(* CODESYS project Pi_Serial_FB_10.project

Project tree, tasks and I/O mapping:
  Device : CODESYS Control for Raspberry Pi SL, 3S - Smart Software Solutions GmbH, version 3.5.12.10
    application Application
      libraries: Standard, * (System); CAA SerialCom, 3.5.12.0 (CAA Technical Workgroup); CAA Types Extern, 3.5.10.0 (CAA Technical Workgroup); CAA Memory, 3.5.12.0 (CAA Technical Workgroup)
      task MainTask (cyclic, interval t#20ms, priority 1) calls PLC_PRG
      task VISU_TASK (cyclic, interval 100 ms, priority 31) calls VisuElems.Visu_Prg
      program PLC_PRG [SFC]: _aInit_active, write_active, read_active, disconnect_active, error_active, Set_COM_active
      visualisation Visualization
      global variables GVL
    SoftMotion General Axis Pool
    I²C
    SPI
      SPI_master : SPI master, 3S - Smart Software Solutions GmbH, version 1.0.0.0
        PiXtend : PiXtend, Qube Solutions UG, version 1.0.0.10
            output Application.GVL.xDO0 : BOOL  // RelayOut.Bit0
            output Application.GVL.byUCControl : BYTE  // CtrlUC
            input  Application.GVL.byUCVersionL : BYTE  // ucVersion_Low
            input  Application.GVL.byUCVersionH : BYTE  // ucVersion_High
            input  Application.GVL.byUCStatus : BYTE  // ucStatus
            unmapped channels: DigIn, GpioIn, AI0, AI1, AI2, AI3, AI0 Raw, AI1 Raw, AI2 Raw, AI3 Raw, Temp0, Temp1, Temp2, Temp3, Humidity0, Humidity1, Humidity2, Humidity3, DigOut, GpioOut, RelayOut, Pwm0, Pwm1, CtrlPwm0, CtrlPwm1, CtrlPwm2, CtrlGpio, CtrlAi0, CtrlAi1, AI Jumpers, DHT11/22
    GPIOs_A_B : GPIOs A/B, 3S - Smart Software Solutions GmbH, version 3.5.11.0
        output rpi_gpio24 : BOOL  // digital outputs (GPIO0..GPIO31).Bit24
        unmapped channels: digital inputs (GPIO0..GPIO31), digital outputs (GPIO0..GPIO31)
    Onewire
    Camera device
      <Empty>
  libraries: VisuSymbols, 3.5.10.0 (System)
  text list GlobalTextList
*)

// Device/Application/GVL
{attribute 'qualified_only'}
VAR_GLOBAL	

	//Digital Outputs
	xDO0: BOOL;
	//Status
	byUCStatus: BYTE;
	byUCVersionL: BYTE;
	byUCVersionH: BYTE;
	//Control
	byUCControl: BYTE;	
END_VAR

// Device/Application/PLC_PRG
PROGRAM PLC_PRG
VAR
	//Visu Variables
	xBtnClear		: BOOL := FALSE;
	xClearAll		: BOOL;	// flag to clear all
	
	//Current State
	iState : INT := 0;

	(* Settings to communicate with the COM Port *)
	aCom1Params : ARRAY [1..7] OF COM.PARAMETER; 
	
	hCom	: CAA.HANDLE; (* handle of the port*)
	como1 	: COM.Open;
	comc1 	: COM.Close;
	comw1 	: COM.Write;
	comr1 	: COM.Read;	
	
	
	sWrite 	: STRING;
	szRead 	: CAA.SIZE;
	uiRead	: UINT;
	
	bReadBuffer	: ARRAY [1..255] OF BYTE; (*Used to read data from the serial port*)
	sReadText	: STRING;
	
	bWriteBuffer: ARRAY [1..255] OF BYTE; (*Used to write data to the serial port*)
	szWrite		: CAA.SIZE;
	
	xReadSuccess	: BOOL;
	xWriteSuccess	: BOOL;
	
	// errors
	xCom1OpenError 	: BOOL;
	xCom1WriteError : BOOL;
	xCom1ReadError 	: BOOL;
	iError			: INT;
	errWrite 		: INT;
	errRead 		: INT;
	Bar				: INT;
	Bar_Temp		: INT;
	
	tTimer			: TON;
	
	sSend 		: STRING(255);	// send message
	sStatus 	: STRING(25);	// status message
	
	//arsReceived : ARRAY[0..1,0..10000] OF STRING(255);	// received messages with timestamp
	Received    :STRING(255);
	intReceived :INT;
	// scrolling
//	iSelect		: INT;			// selected row for scrolling

	iCnt		: INT;
END_VAR

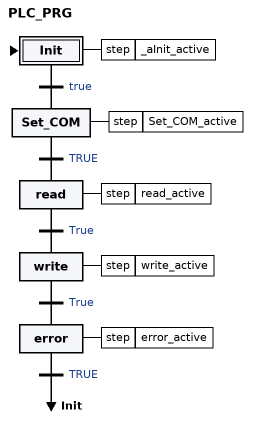
INITIAL_STEP Init:
    _aInit_active(N);  // step action
END_STEP
TRANSITION FROM Init TO Set_COM
    := true;
END_TRANSITION
STEP Set_COM:
    Set_COM_active(N);  // step action
END_STEP
TRANSITION FROM Set_COM TO read
    := TRUE;
END_TRANSITION
STEP read:
    read_active(N);  // step action
END_STEP
TRANSITION FROM read TO write
    := True;
END_TRANSITION
STEP write:
    write_active(N);  // step action
END_STEP
TRANSITION FROM write TO error
    := True;
END_TRANSITION
STEP error:
    error_active(N);  // step action
END_STEP
TRANSITION FROM error TO Init
    := TRUE;
END_TRANSITION

ACTION _aInit_active:

	IF iState = 0 THEN
		 // Init
			sStatus := 'INIT';
			iState:= 5; //Goto 5: Set Parameters	
			IF xClearAll THEN
				// reset errors
				PLC_PRG.xCom1ReadError	:= FALSE;
				PLC_PRG.xCom1WriteError := FALSE;
				PLC_PRG.xCom1OpenError 	:= FALSE;			
				xClearAll := FALSE;
			END_IF
		END_IF
END_ACTION

ACTION write_active:
IF iState = 20 THEN
		
		 // the writing process is started
			sStatus := 'Write';		
			IF NOT comw1.xExecute THEN
				IF Bar = Bar_Temp THEN
					sSend:='g';
				ELSE
					IF Bar = 10 THEN
						sSend:=	'a';
					ELSE	
						sSend:=	INT_TO_STRING(Bar);
					END_IF	
					Bar_Temp:= Bar;
				END_IF	
				szWrite:= INT_TO_UDINT(LEN(sSend));
				// write the string to the buffer for the COM.WRITE Interface
				MEM.MemMove(ADR(sSend), ADR(bWriteBuffer), ANY_TO_UINT(szWrite));
				//sSend := '';	// clear send string
			END_IF
			comw1(xExecute:= TRUE, hCom:= hCom, pBuffer:= ADR(bWriteBuffer), szSize:= szWrite);	// write COM
			// success
			IF comw1.xDone THEN
				comw1(xExecute:= FALSE);	
				xWriteSuccess:= TRUE;
				iState:= 25; // goto 25: Delay after Writing

			ELSIF comw1.xError THEN
				xCom1WriteError:= TRUE;
				iError := comw1.eError;
				errWrite := comw1.eError;
				comw1(xExecute:= FALSE);	
				iState:= 1000;			// error occurred

			END_IF
END_IF
IF iState = 25 THEN 
		
		 // Delay after Writing
			sStatus := 'Write Wait';
			// send or auto send active
			tTimer(IN:= TRUE, PT:= T#250MS);
			IF tTimer.Q THEN
				tTimer(IN:= FALSE);
				xWriteSuccess:= FALSE;	
				iState:= 10;	// Go Back to 10: Read				
			END_IF			
END_IF
END_ACTION

ACTION read_active:
IF iState = 10 THEN
 // Start Reading COM port
		
			IF xClearAll THEN
				// reset errors
				PLC_PRG.xCom1ReadError	:= FALSE;
				PLC_PRG.xCom1WriteError := FALSE;
				PLC_PRG.xCom1OpenError 	:= FALSE;		
				xClearAll := FALSE;
			END_IF
			
			sStatus := 'Read';
			// read COM port
			comr1(xExecute:= TRUE, hCom:= hCom, pBuffer:= ADR(bReadBuffer), szBuffer:= SIZEOF(bReadBuffer));
			IF comr1.xDone THEN
				szRead:= comr1.szSize;
				uiRead:= ANY_TO_UINT(comr1.szSize);
				// check if there is something to read
				IF uiRead > 0 THEN
					// Copy text from the read buffer to sReadText
					MEM.MemMove(ADR(bReadBuffer), ADR(sReadText), uiRead);	// move bReadBuffer to sReadText
					MEM.MemFill(ADR(sReadText) + uiRead, 1, 0);				// write ASCII 000 to byte after received string
					
					IF sReadText <> '' AND sReadText <> 'Uncompressing Li' THEN	// 'Uncrompressing Li' comes from start of Linux and can not be disabled so far
	
						
						//arsReceived[0,iCounter] := GetTime(1);	// get timestamp
						Received := sReadText;	// copy read string to array
						intReceived := STRING_TO_INT(Received);
						sReadText	:= '';						// reset read string
					END_IF
				
					xReadSuccess:= TRUE;
				END_IF
				
				comr1(xExecute:= FALSE);	// Reset xExecute Flag
				iState:= 15; 				// Goto 15: Delay after Reading
			// error
			ELSIF comr1.xError THEN
				xCom1ReadError := TRUE;
				errRead := comr1.eError;
				iError := comr1.eError;
				comr1(xExecute:= FALSE);
				iState:= 1000; // Error occurred
			END_IF
END_IF
IF iState = 15 THEN		
		//Delay after Reading is finished
			sStatus := 'Read Wait';
			xReadSuccess:= FALSE;
			iState := 20; 	// Goto 20: write
END_IF
END_ACTION

ACTION disconnect_active:

END_ACTION

ACTION error_active:
IF iState = 1000 THEN
		 //Error Occurred, go back to 0 after 10 seconds
			sStatus := CONCAT(sStatus,' Error');
			tTimer(IN:= TRUE, PT:= T#10S);
			IF tTimer.Q THEN
				tTimer(IN:= FALSE);
				iState:= 10;
			END_IF			

			
END_IF
END_ACTION

ACTION Set_COM_active:
	//Set COM port parameters
	IF iState = 5 THEN
			sStatus := 'Prepare';
			// port number
			aCom1Params[1].udiParameterId := COM.CAA_Parameter_Constants.udiPort;
			aCom1Params[1].udiValue := 1;
			// baudrate
			aCom1Params[2].udiParameterId := COM.CAA_Parameter_Constants.udiBaudrate;	
			aCom1Params[2].udiValue := 9600;
			// parity
			aCom1Params[3].udiParameterId := COM.CAA_Parameter_Constants.udiParity;
			aCom1Params[3].udiValue := INT_TO_UINT(COM.PARITY.NONE);
			// stopbit
			aCom1Params[4].udiParameterId := COM.CAA_Parameter_Constants.udiStopBits;
			aCom1Params[4].udiValue := INT_TO_UINT(COM.STOPBIT.ONESTOPBIT);
			// timeout
			aCom1Params[5].udiParameterId := COM.CAA_Parameter_Constants.udiTimeout;
			aCom1Params[5].udiValue := 0;
			// byte size
			aCom1Params[6].udiParameterId := COM.CAA_Parameter_Constants.udiByteSize;
			aCom1Params[6].udiValue := 8;
			// mode of transmission
			aCom1Params[7].udiParameterId := COM.CAA_Parameter_Constants.udiBinary;
			aCom1Params[7].udiValue := 0;
			
			// open COM port
			como1(xExecute := TRUE, usiListLength:=UINT_TO_USINT(SIZEOF(aCom1Params)/SIZEOF(COM.PARAMETER)),pParameterList:= ADR(aCom1Params), hCom=> hCom);
			
			// Successful
			IF como1.xDone THEN
				como1(xExecute := FALSE);	// Reset xExecute Flag
				iState := 10; 				// Goto 10: Start Reading
			// Error
			ELSIF como1.xError THEN
				xCom1OpenError := TRUE;
				iError := como1.eError;
				iState := 1000; // Error occurred
			END_IF
	END_IF
END_ACTION

END_PROGRAM

// Device/Application/Visualization
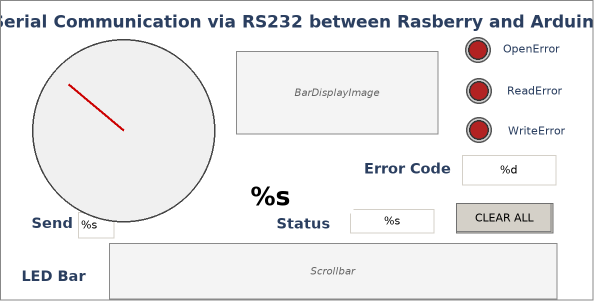
VISUALIZATION Visualization  // 594x301
    Textfield (78,212 36x26), "%s", text variable: PLC_PRG.sSend
        OnMouseClick: write PLC_PRG.sSend via Edit
    Button (456,203 97x30), "CLEAR ALL"
        OnMouseClick: execute { PLC_PRG.xClearAll := TRUE; }
    Textfield (350,209 84x24), "%s", text variable: PLC_PRG.sStatus
    Lamp1 (463,35 30x30), variable: PLC_PRG.xCom1OpenError, style: Lamp-Lamp1-Red
    Label (500,34 63x30), "OpenError"
    Lamp1 (464,76 30x30), variable: PLC_PRG.xCom1ReadError, style: Lamp-Lamp1-Red
    Label (504,76 63x30), "ReadError"
    Label (505,116 63x30), "WriteError"
    Lamp1 (464,115 30x30), variable: PLC_PRG.xCom1WriteError, style: Lamp-Lamp1-Red
    Textfield (462,155 94x30), "%d", text variable: PLC_PRG.iError
    Label (27,208 51x30), "Send"
    Label (5,10 587x23), "Serial Communication via RS232 between Rasberry and Arduino"
    Label (361,156 91x25), "Error Code"
    Label (263,211 81x25), "Status"
    BarDisplayImage (236,51 202x83), value: PLC_PRG.intReceived, style: BarDisplayImage-Gray, scale format: %.1f, scale 15..45
    Scrollbar (109,243 448x56)
        p1057716461: PLC_PRG.Bar
    Label (12,261 83x30), "LED Bar"
    Textfield (188,148 165x65), "%s", tooltip "Temperature", text variable: PLC_PRG.Received
    Meter180 (26,39 195x183), value: PLC_PRG.intReceived, style: Meter-Meter180-Gray, scale format: %.1f, scale 15..45
END_VISUALIZATION
